Omron Sysmac Studio project Treinamento-Sysmac-00 (Sysmac Studio 1.64.0.64008, StandardProject)

# Controller new_Controller_0: NX1P2-9B40DT1 version 1.69
Units and slaves: Node4 : NX-ECC202 (E001); Unit 1 : NX-ID5142-1 (N1); Unit 2 : NX-ID5142-1 (N1_1); Unit 3 : NX-OD5256 (N3); Unit 4 : NX-OD5256 (N3_1)
Task PrimaryTask (priority 4, period or condition 4000): Program0

PROGRAM Program0

(* Section Section0: ladder, written here as Structured Text *)

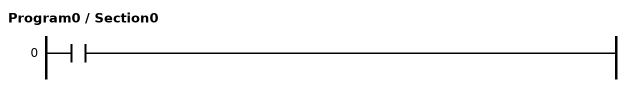
(* Rung 0 *)
END_PROGRAM